// TIA Portal V20 export
// export: Created 2025-12-01T14:57:42.5817105Z, ExportSetting None, DisplayName Totally Integrated Automation Portal, DisplayVersion V20 Update 3, DisplayName TIA Portal Openness, DisplayVersion V20 Update 3, DisplayName TIA Portal Version Control Interface, DisplayVersion V20 Update 3, DisplayName STEP 7 Professional, DisplayVersion V20 Update 3, DisplayName STEP 7 Safety, DisplayVersion V20 Update 2, DisplayName WinCC Basic/Comfort/Advanced, DisplayVersion V20 Update 3, DisplayName WinCC Professional, DisplayVersion V20 Update 3, DisplayName WinCC Unified, DisplayVersion V20 Update 3
FUNCTION "FC9_JDT_Adaptacion" : Void   // FC9, LAD
{ S7_Optimized_Access := 'TRUE' }
// stored: AutoNumber false, SetENOAutomatically false
   VAR_INPUT
      Zona : UInt;   // Numero de Zona
      INP_Pul_TLuces : Bool;
      Jdt_Marcha : Bool;
      JdT_Paro : Bool;
      JdT_Reset : Bool;
      JdT_EmiOK : Bool;
   END_VAR
   VAR_OUTPUT
      L_Verde : Bool;
      L_Naranja : Bool;
      L_Rojo : Bool;
      PLC_Automatico : Bool;
      PLC_Manual : Bool;
      PLC_Marcha : Bool;
      PLC_Paro : Bool;
      PLC_Error : Bool;
      PLC_Reset_OK : Bool;
      PLC_Reset_NOK : Bool;
      PLC_RecepOK : Bool;
   END_VAR
   VAR_IN_OUT
      CodigoError : Word;
   END_VAR
   VAR_TEMP
      MesaEnError : UInt;
   END_VAR
BEGIN

NETWORK
TITLE = INICIALIZAR

NETWORK
TITLE = CODIGO DE ERROR - DE ZONA
/////////////////////////////////////////////////////////////////////////////////////
////////////////////////////////////////////////////////////////////////////////////
////////////////////////////////////////////////////////////////////////////////////
/// --- Codigo de Error De Zona Dos Digitos -- 9x EE
      L     0;  // Inicializa el Codigo de Error
      T     #CodigoError;

      SET;  // Existe Error de Zona ?
      AN    "DB840_Emision".DispoArmario[#Zona].Protocolo.Error;
      JC    Final_ErrorDeZona;

/// --- Primer Digito - Error
      L     "DB840_Emision".DispoArmario[#Zona].Error;
      L     10;
      MOD;
      T     #CodigoError;

/// --- Segundo Digito - Error
      L     "DB840_Emision".DispoArmario[#Zona].Error;
      L     10;
      /D;
      L     10;
      MOD;
      SLD   4;
      L     #CodigoError;
      OW;
      T     #CodigoError;

/// --- Tercer Digito - Numero de Zona
      L     #Zona;
      SLD   8;
      L     #CodigoError;
      OW;
      T     #CodigoError;

/// --- Cuarto Digito - Indicacion De Zona
      L     w#16#9000;
      L     #CodigoError;
      OW;
      T     #CodigoError;

/// --- Final de Codificacion del Error de Zona
Final_ErrorDeZona:NOP   0;



NETWORK
TITLE = CODIGO DE ERROR - DE MESA
/////////////////////////////////////////////////////////////////////////////////////
////////////////////////////////////////////////////////////////////////////////////
////////////////////////////////////////////////////////////////////////////////////
/// --- Codigo de Error De Mesa -- 6 MMMM
      SET;  // Existe Error de Zona ?
      A     "DB840_Emision".DispoArmario[#Zona].Protocolo.Error;
      JC    Final_ErrorDeMesa;

      SET;  // Existe Error de Mesa ?
      AN    "DB901_Estado_Zonas".EstadoZona[#Zona].VariablesInternas.MesasError;
      JC    Final_ErrorDeMesa;

/// --- Numero de Mesa en Error
      L     0;
      T     #MesaEnError;
InicioBucle_BusquedaDeMesaEnError:NOP   0;
      L     "CTE_MaxMesas";  // - Final del Numero de Mesas ?
      L     #MesaEnError;
      <=I;
      JC    FinalBucle_BusquedaDeMesaEnError;

      L     #MesaEnError;
      L     1;
      +I;
      T     #MesaEnError;

      SET;  /// Mesa de la Zona (0)
      L     #Zona;
      L     "DB914_Conf_Mesas_DeZona".MesasDeZona[#MesaEnError, 0].ZonaPerteneceMesa;
      ==I;
      JC    MesaEncontrada_BusquedaDeMEsaEnError;

      SET;  /// Mesa de la Zona (1)
      L     #Zona;
      L     "DB914_Conf_Mesas_DeZona".MesasDeZona[#MesaEnError, 1].ZonaPerteneceMesa;
      ==I;
      JC    MesaEncontrada_BusquedaDeMEsaEnError;

      SET;  /// Mesa de la Zona (2)
      L     #Zona;
      L     "DB914_Conf_Mesas_DeZona".MesasDeZona[#MesaEnError, 2].ZonaPerteneceMesa;
      ==I;
      JC    MesaEncontrada_BusquedaDeMEsaEnError;

      SET;  /// Mesa de la Zona (3)
      L     #Zona;
      L     "DB914_Conf_Mesas_DeZona".MesasDeZona[#MesaEnError, 3].ZonaPerteneceMesa;
      ==I;
      JC    MesaEncontrada_BusquedaDeMEsaEnError;

      SET;  /// Mesa de la Zona (4)
      L     #Zona;
      L     "DB914_Conf_Mesas_DeZona".MesasDeZona[#MesaEnError, 4].ZonaPerteneceMesa;
      ==I;
      JC    MesaEncontrada_BusquedaDeMEsaEnError;

      JU    InicioBucle_BusquedaDeMesaEnError;

MesaEncontrada_BusquedaDeMEsaEnError:NOP   0;
      SET;  // - Mesa o Maquina en Error
      A     "DB902_Estado_ZonaMesa".EstadoMesas[#MesaEnError].Error_CBx;
      O     "DB903_Estado_ZonaMaquina".EstadoMaquina[#MesaEnError].Error_CBx;
      JC    FinalBucle_BusquedaDeMesaEnError;

      JU    InicioBucle_BusquedaDeMesaEnError;

////////////////////////////////////////////////////////////////////////////////////
FinalBucle_BusquedaDeMesaEnError:NOP   0;

/// --- Primer Digito - Mesa
      L     #MesaEnError;
      L     10;
      MOD;
      T     #CodigoError;

/// --- Segundo Digito - Mesa
      L     #MesaEnError;
      L     10;
      /D;
      L     10;
      MOD;
      SLD   4;
      L     #CodigoError;
      OW;
      T     #CodigoError;

/// --- Tercer Digito - Mesa
      L     #MesaEnError;
      L     100;
      /D;
      L     10;
      MOD;
      SLD   8;
      L     #CodigoError;
      OW;
      T     #CodigoError;

/// --- Cuarto Digito - Indicacion De Mesa
      L     w#16#6000;
      L     #CodigoError;
      OW;
      T     #CodigoError;

/// --- Final de Codificacion del Error de Zona
Final_ErrorDeMesa:NOP   0;



NETWORK
TITLE = EMISION DE LA ZONA
/////////////////////////////////////////////////////////////////////////////////////
////////////////////////////////////////////////////////////////////////////////////
////////////////////////////////////////////////////////////////////////////////////
/// --- COMPROBAR si esta con el JdT Antiguo
      SET;
      AN    "Activar_JdTAntiguo";
      JC    Final_EmisionZona;


/////////////////////////////////////////////////////////////////////////////////////
////////////////////////////////////////////////////////////////////////////////////
////////////////////////////////////////////////////////////////////////////////////
/// --- Automatico / Manual
      SET;
      A     "DB840_Emision".DispoArmario[#Zona].Protocolo.Automatico;
      =     #PLC_Automatico;
      SET;
      A     "DB840_Emision".DispoArmario[#Zona].Protocolo.Manual;
      =     #PLC_Manual;


/////////////////////////////////////////////////////////////////////////////////////
////////////////////////////////////////////////////////////////////////////////////
////////////////////////////////////////////////////////////////////////////////////
/// --- Marcha / Paro / ErrorPLC
      SET;
      A     "DB840_Emision".DispoArmario[#Zona].Protocolo.Marcha;
      =     #PLC_Marcha;
      SET;
      A     "DB840_Emision".DispoArmario[#Zona].Protocolo.Paro;
      =     #PLC_Paro;
      SET;
      A     "DB840_Emision".DispoArmario[#Zona].Protocolo.Error;
      O     "DB901_Estado_Zonas".EstadoZona[#Zona].VariablesInternas.MesasError;
      =     #PLC_Error;

/////////////////////////////////////////////////////////////////////////////////////
////////////////////////////////////////////////////////////////////////////////////
////////////////////////////////////////////////////////////////////////////////////
/// --- Reset
      SET;
      A     "DB840_Emision".DispoArmario[#Zona].Protocolo.ResetOK;
      =     #PLC_Reset_OK;
      SET;
      A     "DB840_Emision".DispoArmario[#Zona].Protocolo.ResetNOK;
      =     #PLC_Reset_NOK;

/////////////////////////////////////////////////////////////////////////////////////
////////////////////////////////////////////////////////////////////////////////////
////////////////////////////////////////////////////////////////////////////////////
/// --- Comunicacion
      SET;
      A     "DB840_Emision".DispoArmario[#Zona].Protocolo.RecepOK;
      =     #PLC_RecepOK;


/////////////////////////////////////////////////////////////////////////////////////
////////////////////////////////////////////////////////////////////////////////////
////////////////////////////////////////////////////////////////////////////////////
/// --- FINAL de la EMISION DE LA ZONA
Final_EmisionZona:NOP   0;



NETWORK
TITLE = RECEPCION DE LA ZONA
/////////////////////////////////////////////////////////////////////////////////////
////////////////////////////////////////////////////////////////////////////////////
////////////////////////////////////////////////////////////////////////////////////
/// --- COMPROBAR si esta con el JdT Antiguo
      SET;
      AN    "Activar_JdTAntiguo";
      JC    Final_RecepcionZona;


/////////////////////////////////////////////////////////////////////////////////////
/////////////////////////////////////////////////////////////////////////////////////
/////////////////////////////////////////////////////////////////////////////////////
/// --- Ordenes
      SET;
      A     #Jdt_Marcha;
      =     "DB841_Recepcion".DispoArmario[#Zona].Protocolo.Marcha;
      SET;
      A     #JdT_Paro;
      =     "DB841_Recepcion".DispoArmario[#Zona].Protocolo.Paro;
      SET;
      A     #JdT_Reset;
      =     "DB841_Recepcion".DispoArmario[#Zona].Protocolo.Reset;

/////////////////////////////////////////////////////////////////////////////////////
////////////////////////////////////////////////////////////////////////////////////
////////////////////////////////////////////////////////////////////////////////////
/// --- Comunicacion
      SET;
      A     #JdT_EmiOK;
      =     "DB841_Recepcion".DispoArmario[#Zona].Protocolo.EmiOK;


/////////////////////////////////////////////////////////////////////////////////////
////////////////////////////////////////////////////////////////////////////////////
////////////////////////////////////////////////////////////////////////////////////
/// --- FINAL de la RECEPCION DE LA ZONA
Final_RecepcionZona:NOP   0;



REGION Network 6: SALIDAS - Baliza VERDE
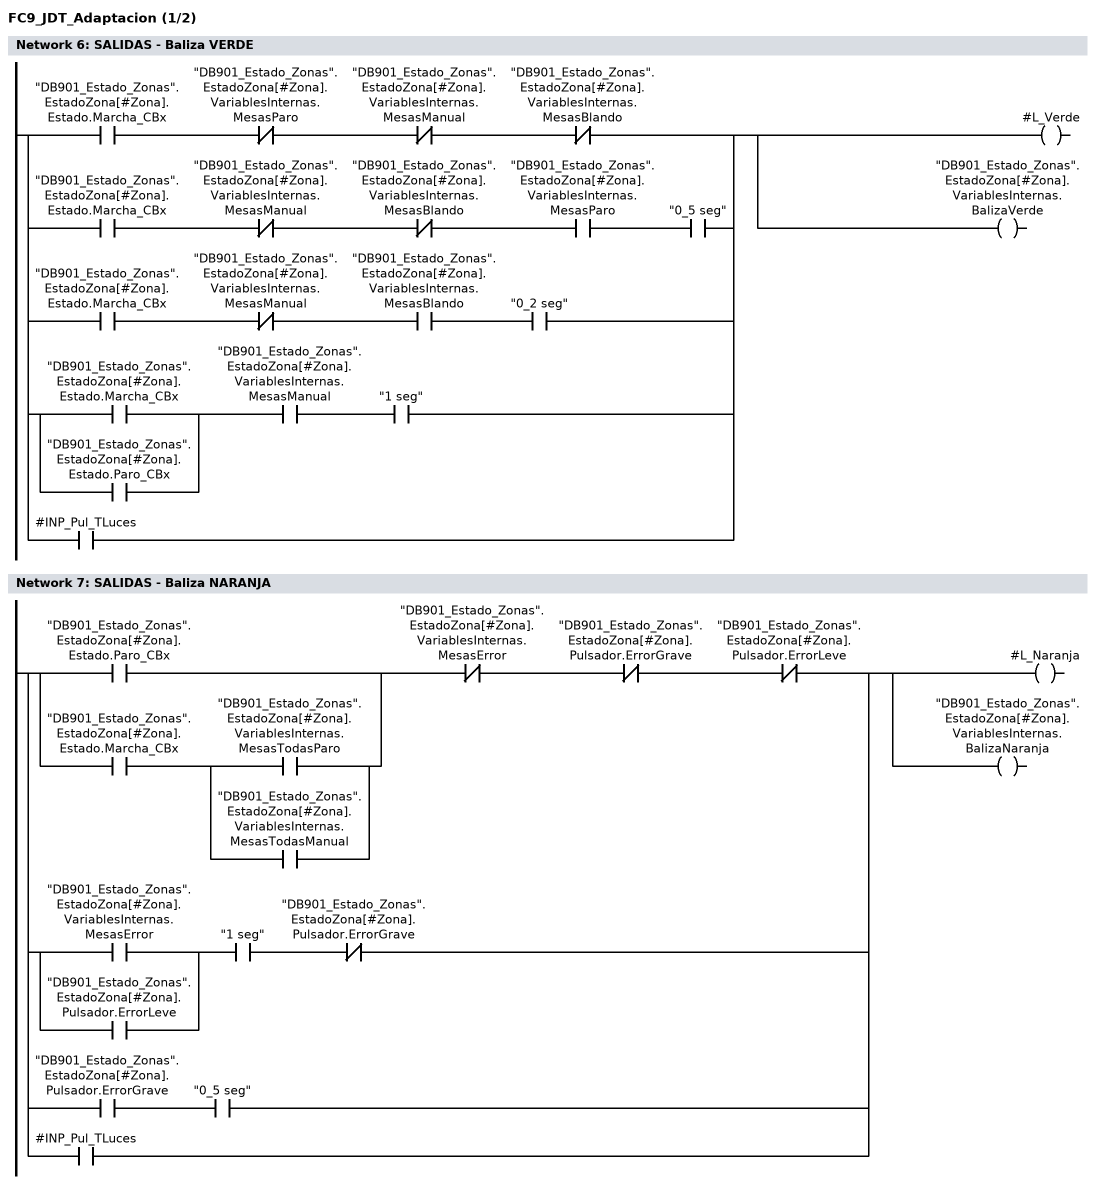
   RUNG wire#powerrail
      Contact( "DB901_Estado_Zonas".EstadoZona[#Zona].Estado.Marcha_CBx )
      I_Contact( "DB901_Estado_Zonas".EstadoZona[#Zona].VariablesInternas.MesasParo )
      I_Contact( "DB901_Estado_Zonas".EstadoZona[#Zona].VariablesInternas.MesasManual )
      I_Contact( "DB901_Estado_Zonas".EstadoZona[#Zona].VariablesInternas.MesasBlando )
      wire#w1
      Coil( #L_Verde )
   END_RUNG
   RUNG wire#powerrail
      Contact( "DB901_Estado_Zonas".EstadoZona[#Zona].Estado.Marcha_CBx )
      I_Contact( "DB901_Estado_Zonas".EstadoZona[#Zona].VariablesInternas.MesasManual )
      I_Contact( "DB901_Estado_Zonas".EstadoZona[#Zona].VariablesInternas.MesasBlando )
      Contact( "DB901_Estado_Zonas".EstadoZona[#Zona].VariablesInternas.MesasParo )
      Contact( "0_5 seg" )
   END_RUNG wire#w1
   RUNG wire#powerrail
      Contact( "DB901_Estado_Zonas".EstadoZona[#Zona].Estado.Marcha_CBx )
      I_Contact( "DB901_Estado_Zonas".EstadoZona[#Zona].VariablesInternas.MesasManual )
      Contact( "DB901_Estado_Zonas".EstadoZona[#Zona].VariablesInternas.MesasBlando )
      Contact( "0_2 seg" )
   END_RUNG wire#w1
   RUNG wire#powerrail
      Contact( "DB901_Estado_Zonas".EstadoZona[#Zona].Estado.Marcha_CBx )
      wire#w2
      Contact( "DB901_Estado_Zonas".EstadoZona[#Zona].VariablesInternas.MesasManual )
      Contact( "1 seg" )
   END_RUNG wire#w1
   RUNG wire#powerrail
      Contact( "DB901_Estado_Zonas".EstadoZona[#Zona].Estado.Paro_CBx )
   END_RUNG wire#w2
   RUNG wire#powerrail
      Contact( #INP_Pul_TLuces )
   END_RUNG wire#w1
   RUNG wire#w1
      Coil( "DB901_Estado_Zonas".EstadoZona[#Zona].VariablesInternas.BalizaVerde )
   END_RUNG
   // the same network as SCL:
   #L_Verde := ("DB901_Estado_Zonas".EstadoZona[#Zona].Estado.Marcha_CBx AND NOT "DB901_Estado_Zonas".EstadoZona[#Zona].VariablesInternas.MesasParo AND NOT "DB901_Estado_Zonas".EstadoZona[#Zona].VariablesInternas.MesasManual AND NOT "DB901_Estado_Zonas".EstadoZona[#Zona].VariablesInternas.MesasBlando) OR ("DB901_Estado_Zonas".EstadoZona[#Zona].Estado.Marcha_CBx AND NOT "DB901_Estado_Zonas".EstadoZona[#Zona].VariablesInternas.MesasManual AND NOT "DB901_Estado_Zonas".EstadoZona[#Zona].VariablesInternas.MesasBlando AND "DB901_Estado_Zonas".EstadoZona[#Zona].VariablesInternas.MesasParo AND "0_5 seg") OR ("DB901_Estado_Zonas".EstadoZona[#Zona].Estado.Marcha_CBx AND NOT "DB901_Estado_Zonas".EstadoZona[#Zona].VariablesInternas.MesasManual AND "DB901_Estado_Zonas".EstadoZona[#Zona].VariablesInternas.MesasBlando AND "0_2 seg") OR (("DB901_Estado_Zonas".EstadoZona[#Zona].Estado.Marcha_CBx OR "DB901_Estado_Zonas".EstadoZona[#Zona].Estado.Paro_CBx) AND "DB901_Estado_Zonas".EstadoZona[#Zona].VariablesInternas.MesasManual AND "1 seg") OR #INP_Pul_TLuces;
   "DB901_Estado_Zonas".EstadoZona[#Zona].VariablesInternas.BalizaVerde := #L_Verde;
END_REGION

REGION Network 7: SALIDAS - Baliza NARANJA
   RUNG wire#powerrail
      Contact( "DB901_Estado_Zonas".EstadoZona[#Zona].Estado.Paro_CBx )
      wire#w1
      I_Contact( "DB901_Estado_Zonas".EstadoZona[#Zona].VariablesInternas.MesasError )
      I_Contact( "DB901_Estado_Zonas".EstadoZona[#Zona].Pulsador.ErrorGrave )
      I_Contact( "DB901_Estado_Zonas".EstadoZona[#Zona].Pulsador.ErrorLeve )
      wire#w3
      Coil( #L_Naranja )
   END_RUNG
   RUNG wire#powerrail
      Contact( "DB901_Estado_Zonas".EstadoZona[#Zona].Estado.Marcha_CBx )
      wire#w2
      Contact( "DB901_Estado_Zonas".EstadoZona[#Zona].VariablesInternas.MesasTodasParo )
   END_RUNG wire#w1
   RUNG wire#w2
      Contact( "DB901_Estado_Zonas".EstadoZona[#Zona].VariablesInternas.MesasTodasManual )
   END_RUNG wire#w1
   RUNG wire#powerrail
      Contact( "DB901_Estado_Zonas".EstadoZona[#Zona].VariablesInternas.MesasError )
      wire#w4
      Contact( "1 seg" )
      I_Contact( "DB901_Estado_Zonas".EstadoZona[#Zona].Pulsador.ErrorGrave )
   END_RUNG wire#w3
   RUNG wire#powerrail
      Contact( "DB901_Estado_Zonas".EstadoZona[#Zona].Pulsador.ErrorLeve )
   END_RUNG wire#w4
   RUNG wire#powerrail
      Contact( "DB901_Estado_Zonas".EstadoZona[#Zona].Pulsador.ErrorGrave )
      Contact( "0_5 seg" )
   END_RUNG wire#w3
   RUNG wire#powerrail
      Contact( #INP_Pul_TLuces )
   END_RUNG wire#w3
   RUNG wire#w3
      Coil( "DB901_Estado_Zonas".EstadoZona[#Zona].VariablesInternas.BalizaNaranja )
   END_RUNG
   // the same network as SCL:
   #L_Naranja := (("DB901_Estado_Zonas".EstadoZona[#Zona].Estado.Paro_CBx OR ("DB901_Estado_Zonas".EstadoZona[#Zona].Estado.Marcha_CBx AND ("DB901_Estado_Zonas".EstadoZona[#Zona].VariablesInternas.MesasTodasParo OR "DB901_Estado_Zonas".EstadoZona[#Zona].VariablesInternas.MesasTodasManual))) AND NOT "DB901_Estado_Zonas".EstadoZona[#Zona].VariablesInternas.MesasError AND NOT "DB901_Estado_Zonas".EstadoZona[#Zona].Pulsador.ErrorGrave AND NOT "DB901_Estado_Zonas".EstadoZona[#Zona].Pulsador.ErrorLeve) OR (("DB901_Estado_Zonas".EstadoZona[#Zona].VariablesInternas.MesasError OR "DB901_Estado_Zonas".EstadoZona[#Zona].Pulsador.ErrorLeve) AND "1 seg" AND NOT "DB901_Estado_Zonas".EstadoZona[#Zona].Pulsador.ErrorGrave) OR ("DB901_Estado_Zonas".EstadoZona[#Zona].Pulsador.ErrorGrave AND "0_5 seg") OR #INP_Pul_TLuces;
   "DB901_Estado_Zonas".EstadoZona[#Zona].VariablesInternas.BalizaNaranja := #L_Naranja;
END_REGION

REGION Network 8: SALIDAS - Baliza ROJA
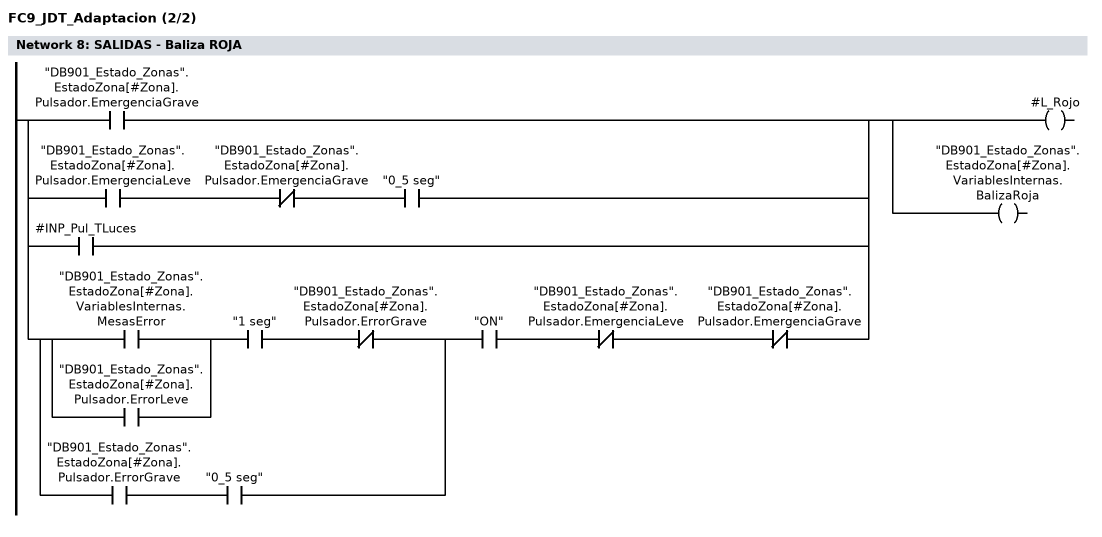
   RUNG wire#powerrail
      Contact( "DB901_Estado_Zonas".EstadoZona[#Zona].Pulsador.EmergenciaGrave )
      wire#w1
      Coil( #L_Rojo )
   END_RUNG
   RUNG wire#powerrail
      Contact( "DB901_Estado_Zonas".EstadoZona[#Zona].Pulsador.EmergenciaLeve )
      I_Contact( "DB901_Estado_Zonas".EstadoZona[#Zona].Pulsador.EmergenciaGrave )
      Contact( "0_5 seg" )
   END_RUNG wire#w1
   RUNG wire#powerrail
      Contact( #INP_Pul_TLuces )
   END_RUNG wire#w1
   RUNG wire#powerrail
      Contact( "DB901_Estado_Zonas".EstadoZona[#Zona].VariablesInternas.MesasError )
      wire#w2
      Contact( "1 seg" )
      I_Contact( "DB901_Estado_Zonas".EstadoZona[#Zona].Pulsador.ErrorGrave )
      wire#w3
      Contact( "ON" )
      I_Contact( "DB901_Estado_Zonas".EstadoZona[#Zona].Pulsador.EmergenciaLeve )
      I_Contact( "DB901_Estado_Zonas".EstadoZona[#Zona].Pulsador.EmergenciaGrave )
   END_RUNG wire#w1
   RUNG wire#powerrail
      Contact( "DB901_Estado_Zonas".EstadoZona[#Zona].Pulsador.ErrorLeve )
   END_RUNG wire#w2
   RUNG wire#powerrail
      Contact( "DB901_Estado_Zonas".EstadoZona[#Zona].Pulsador.ErrorGrave )
      Contact( "0_5 seg" )
   END_RUNG wire#w3
   RUNG wire#w1
      Coil( "DB901_Estado_Zonas".EstadoZona[#Zona].VariablesInternas.BalizaRoja )
   END_RUNG
   // the same network as SCL:
   #L_Rojo := "DB901_Estado_Zonas".EstadoZona[#Zona].Pulsador.EmergenciaGrave OR ("DB901_Estado_Zonas".EstadoZona[#Zona].Pulsador.EmergenciaLeve AND NOT "DB901_Estado_Zonas".EstadoZona[#Zona].Pulsador.EmergenciaGrave AND "0_5 seg") OR #INP_Pul_TLuces OR (((("DB901_Estado_Zonas".EstadoZona[#Zona].VariablesInternas.MesasError OR "DB901_Estado_Zonas".EstadoZona[#Zona].Pulsador.ErrorLeve) AND "1 seg" AND NOT "DB901_Estado_Zonas".EstadoZona[#Zona].Pulsador.ErrorGrave) OR ("DB901_Estado_Zonas".EstadoZona[#Zona].Pulsador.ErrorGrave AND "0_5 seg")) AND "ON" AND NOT "DB901_Estado_Zonas".EstadoZona[#Zona].Pulsador.EmergenciaLeve AND NOT "DB901_Estado_Zonas".EstadoZona[#Zona].Pulsador.EmergenciaGrave);
   "DB901_Estado_Zonas".EstadoZona[#Zona].VariablesInternas.BalizaRoja := #L_Rojo;
END_REGION
END_FUNCTION
